Staubli VAL3: remErrZone.pgx

program remErrZone(string& sReturn[] (dimensions=1))
  local string sErr
begin
  // Error raised when robot enters a stay clear zone
  // Add to buffer instead of sending to IOC immediately
  //
  logMsg("call remErrZone")
  sErr="301: Entered STAY CLEAR zone!"
  call remErrBufferAdd(sErr)
  putln("ERROR "+sErr)
  logMsg("ERROR "+sErr)
  sReturn=""
end
